// The root's instance DB name IS its browse name (Part IV s.3.10.1, s.4.8):
// OPC UA path <PLC>/DataBlocksInstance/SpikeUnit/...,
// GetInstancePath => '"SpikeUnit"', children '"SpikeUnit".CylA'.
DATA_BLOCK "SpikeUnit"
{ S7_Optimized_Access := 'TRUE' }
VERSION : 0.1
NON_RETAIN
"FB_SpkUnit"

BEGIN

END_DATA_BLOCK
